FUNCTION alg_g_w_W2: REAL
{ S7_Optimized_Access := 'false' }
    VAR_INPUT
        state: STATE;
    END_VAR

BEGIN
    alg_g_w_W2 := state.curTime;
END_FUNCTION
